(* PLC project Generated.project, CODESYS CODESYS V3.5 SP19 Patch 1 *)
(* stored: creationDateTime 2026-09-06T13:00:42.569534, modificationDateTime 2026-09-06T13:00:42.569534 *)

(* ═══════════════════════════════════════════════════════════════ 🚨 ST_AlarmBanner — Bandeau d'alarme defilant (carrousel n/N) ─────────────────────────────────────────────────────────────── 🎯 Role : liste les defauts/warnings actifs de toute la machine, affiches un a la fois en rotation (FB_Hmi_BannerFormatter S5) 📄 Doc : DOC/AF/AF_Partie-07_Interface_IHM_v2.3.md S6 ═══════════════════════════════════════════════════════════════ *)
TYPE ST_AlarmBanner : STRUCT
  HasAlarm : BOOL;  (* TRUE = au moins un defaut/warning actif *)
  Text : STRING(120);  (* Texte du message courant : [ORGANE] raison breve *)
  Index : INT;  (* Position courante (1-based, 0 si aucun defaut) *)
  Count : INT;  (* Nombre total de messages actifs *)
  AlarmArray : ARRAY[0..49] OF STRING(120);  (* 📋 Liste complete instantanee de tous les defauts actifs *)
END_STRUCT;
END_TYPE
